(* CODESYS project Lark_Lubrication_AnandFeed.project
   Title: Lark_Lubrication_AnandFeed
   Version: 0.0.0.0

Project tree, tasks and I/O mapping:
  MyController : TM218LDA24DRN, Schneider Electric, order no. TM218LDA24DRN, version 4.0.1.26
    application Application
      libraries: Standard, * (System)
      task MAST (cyclic, interval 20 ms, priority 15, watchdog 100 ms x 1) calls POU
      function HiddenPOU [ST]
      global variables GVL
      program POU [FBD]
    Embedded Functions
      IO : IO, Schneider Electric, version 4.0.1.26
          input  iwIO_IW0 : WORD  // IW0
          input  Motor_Trip : BOOL  // IW0.I0
          input  Motor_ON_FB : BOOL  // IW0.I1
          input  Manual_Start : BOOL  // IW0.I2
          input  Manual_Stop : BOOL  // IW0.I3
          input  Manual_SS : BOOL  // IW0.I4
          input  Line2_SS : BOOL  // IW0.I5
          input  Tank_Empty_LS : BOOL  // IW0.I6
          input  Sensor1 : BOOL  // IW0.I7
          input  Sensor2 : BOOL  // IW0.I8
          output Motor_ON_CMD : BOOL  // QW0.Q0
          output Valve_On : BOOL  // QW0.Q3
          unmapped channels: QW0
      HSC : HSC, Schneider Electric, version 4.0.1.26
    Serial Line 1
      SoMachine_Network_Manager : SoMachine-Network Manager, Schneider Electric, version 4.0.0.2
    Serial Line 2
      Modbus_Manager : Modbus Manager, Schneider Electric, version 4.0.0.2
*)

// MyController/Application/GVL
VAR_GLOBAL
	
	Line1_On_Actual_Time AT %MD4 : DINT;
	Line1_Interval_Actual_Time AT %MD5 : DINT;
	
	Line2_On_Actual_Time AT %MD6 : DINT;
	Line2_Interval_Actual_Time AT %MD7 : DINT;
	
	Motor_Trip_IND AT %MX100.7: BOOL;
	Motor_On_IND AT %MX100.2: BOOL;
	Line1_On_CMD AT %MX100.4: BOOL;
	Line2_On_CMD AT %MX100.5: BOOL;
	Auto_SS AT %MX100.3: BOOL;
	TankEmptyLS_HMI AT %MX100.6: BOOL;
END_VAR

VAR_GLOBAL RETAIN
	Line1_SetTime AT %MD0 : DINT;
	Line1_IntervalTime AT %MD1 : DINT;
	
	Line2_SetTime AT %MD2 : DINT;
	Line2_IntervalTime AT %MD3 : DINT;
	
	Line1_Selected AT %MX100.0 : BOOL;
	Line2_Selected AT %MX100.1 : BOOL;
END_VAR

// MyController/Application/POU
PROGRAM POU
VAR
	TON_0: TON;
	SR_0: SR;
	R_TRIG_0: R_TRIG;
	SR_1: SR;
	Line1ON: BOOL;
	TON_1: TON;
	line1_SetTime_TIME: TIME;
	line1_On_ET_TIME: TIME;
	line1On_Elapsed: BOOL;
	line1_IntervalTime_TIME: TIME;
	line1_Int_ET_TIME: TIME;
	line1_Repeat: BOOL;
	RS_0: RS;
	Line2ON: BOOL;
	R_TRIG_1: R_TRIG;
	RS_1: RS;
	line2_Repeat: BOOL;
	TON_2: TON;
	line2_SetTime_TIME: TIME;
	line2_On_ET_TIME: TIME;
	line2On_Elapsed: BOOL;
	SR_2: SR;
	TON_3: TON;
	line2_IntervalTime_TIME: TIME;
	line2_Int_ET_TIME: TIME;
	RS_2: RS;
	Start_CMD: BOOL;
	Motor_ON_CMD_1: BOOL;
	Motor_ON_CMD_2: BOOL;
	TON_4: TON;
	test: BOOL;
END_VAR
VAR // added by the converter: edge detectors and wires of the graphical bodies
    _w1, _w2, _w3 : BOOL;
END_VAR

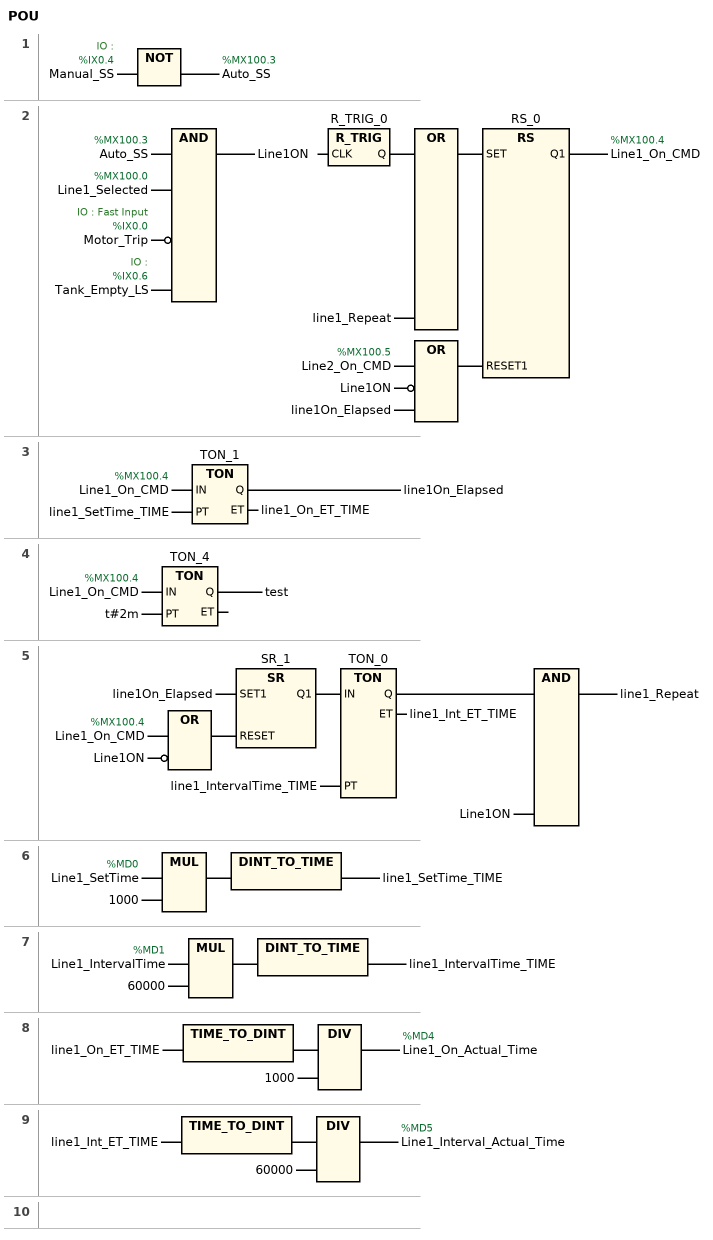
// NETWORK 1
//   Manual_SS: IO : | AT %IX0.4
//   Auto_SS: AT %MX100.3
Auto_SS := NOT Manual_SS;

// NETWORK 2
//   Auto_SS: AT %MX100.3
//   Line1_Selected: AT %MX100.0
//   Motor_Trip: IO : Fast Input | AT %IX0.0
//   Tank_Empty_LS: IO : | AT %IX0.6
//   Line2_On_CMD: AT %MX100.5
//   Line1_On_CMD: AT %MX100.4
_w1 := Auto_SS AND Line1_Selected AND NOT Motor_Trip AND Tank_Empty_LS;
Line1ON := _w1;
R_TRIG_0(CLK := _w1); // R_TRIG
RS_0(SET := R_TRIG_0.Q OR line1_Repeat, RESET1 := Line2_On_CMD OR NOT Line1ON OR line1On_Elapsed); // RS
Line1_On_CMD := RS_0.Q1;

// NETWORK 3
//   Line1_On_CMD: AT %MX100.4
TON_1(IN := Line1_On_CMD, PT := line1_SetTime_TIME, ET => line1_On_ET_TIME); // TON
line1On_Elapsed := TON_1.Q;

// NETWORK 4
//   Line1_On_CMD: AT %MX100.4
TON_4(IN := Line1_On_CMD, PT := t#2m); // TON
test := TON_4.Q;

// NETWORK 5
//   Line1_On_CMD: AT %MX100.4
SR_1(SET1 := line1On_Elapsed, RESET := Line1_On_CMD OR NOT Line1ON); // SR
TON_0(IN := SR_1.Q1, PT := line1_IntervalTime_TIME, ET => line1_Int_ET_TIME); // TON
line1_Repeat := TON_0.Q AND Line1ON;

// NETWORK 6
//   Line1_SetTime: AT %MD0
line1_SetTime_TIME := DINT_TO_TIME(Line1_SetTime * 1000);

// NETWORK 7
//   Line1_IntervalTime: AT %MD1
line1_IntervalTime_TIME := DINT_TO_TIME(Line1_IntervalTime * 60000);

// NETWORK 8
//   Line1_On_Actual_Time: AT %MD4
Line1_On_Actual_Time := TIME_TO_DINT(line1_On_ET_TIME) / 1000;

// NETWORK 9
//   Line1_Interval_Actual_Time: AT %MD5
Line1_Interval_Actual_Time := TIME_TO_DINT(line1_Int_ET_TIME) / 60000;

// NETWORK 10

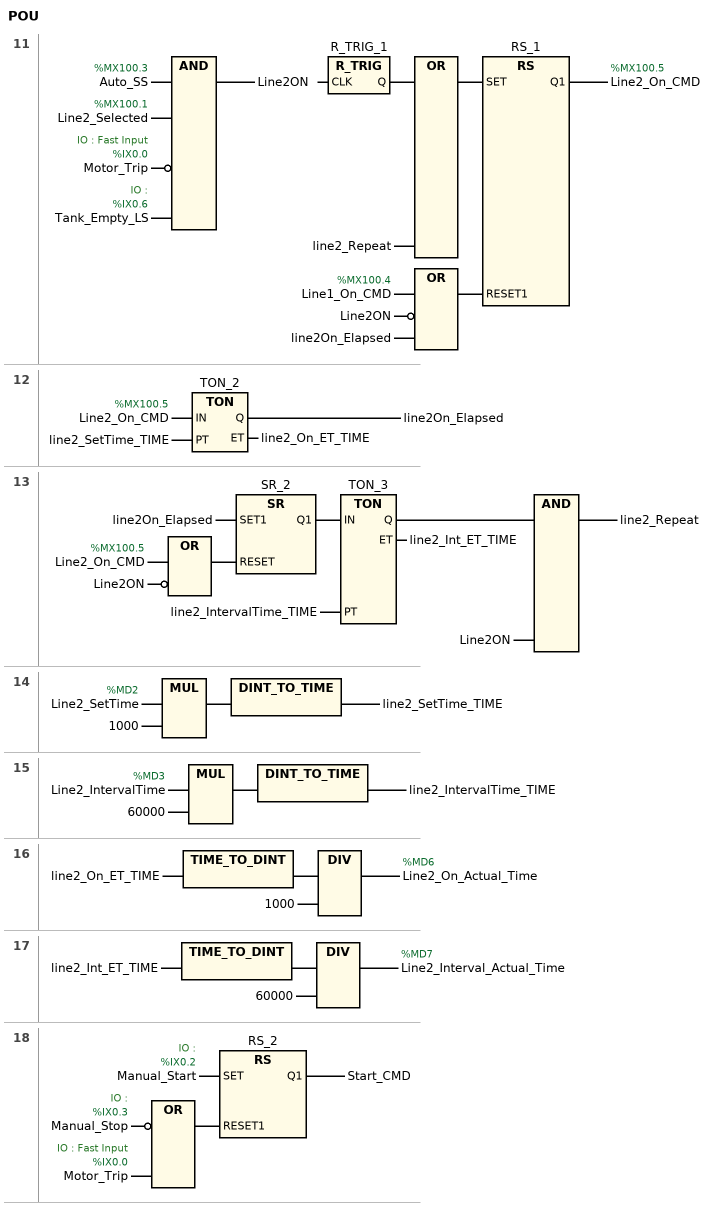
// NETWORK 11
//   Auto_SS: AT %MX100.3
//   Line2_Selected: AT %MX100.1
//   Motor_Trip: IO : Fast Input | AT %IX0.0
//   Tank_Empty_LS: IO : | AT %IX0.6
//   Line1_On_CMD: AT %MX100.4
//   Line2_On_CMD: AT %MX100.5
_w2 := Auto_SS AND Line2_Selected AND NOT Motor_Trip AND Tank_Empty_LS;
Line2ON := _w2;
R_TRIG_1(CLK := _w2); // R_TRIG
RS_1(SET := R_TRIG_1.Q OR line2_Repeat, RESET1 := Line1_On_CMD OR NOT Line2ON OR line2On_Elapsed); // RS
Line2_On_CMD := RS_1.Q1;

// NETWORK 12
//   Line2_On_CMD: AT %MX100.5
TON_2(IN := Line2_On_CMD, PT := line2_SetTime_TIME, ET => line2_On_ET_TIME); // TON
line2On_Elapsed := TON_2.Q;

// NETWORK 13
//   Line2_On_CMD: AT %MX100.5
SR_2(SET1 := line2On_Elapsed, RESET := Line2_On_CMD OR NOT Line2ON); // SR
TON_3(IN := SR_2.Q1, PT := line2_IntervalTime_TIME, ET => line2_Int_ET_TIME); // TON
line2_Repeat := TON_3.Q AND Line2ON;

// NETWORK 14
//   Line2_SetTime: AT %MD2
line2_SetTime_TIME := DINT_TO_TIME(Line2_SetTime * 1000);

// NETWORK 15
//   Line2_IntervalTime: AT %MD3
line2_IntervalTime_TIME := DINT_TO_TIME(Line2_IntervalTime * 60000);

// NETWORK 16
//   Line2_On_Actual_Time: AT %MD6
Line2_On_Actual_Time := TIME_TO_DINT(line2_On_ET_TIME) / 1000;

// NETWORK 17
//   Line2_Interval_Actual_Time: AT %MD7
Line2_Interval_Actual_Time := TIME_TO_DINT(line2_Int_ET_TIME) / 60000;

// NETWORK 18
//   Manual_Start: IO : | AT %IX0.2
//   Manual_Stop: IO : | AT %IX0.3
//   Motor_Trip: IO : Fast Input | AT %IX0.0
RS_2(SET := Manual_Start, RESET1 := NOT Manual_Stop OR Motor_Trip); // RS
Start_CMD := RS_2.Q1;

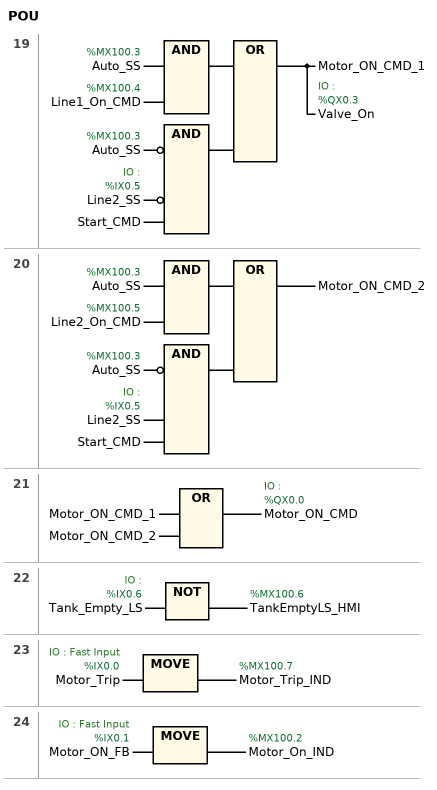
// NETWORK 19
//   Auto_SS: AT %MX100.3
//   Line1_On_CMD: AT %MX100.4
//   Line2_SS: IO : | AT %IX0.5
//   Valve_On: IO : | AT %QX0.3
_w3 := Auto_SS AND Line1_On_CMD OR NOT Auto_SS AND NOT Line2_SS AND Start_CMD;
Motor_ON_CMD_1 := _w3;
Valve_On := _w3;

// NETWORK 20
//   Auto_SS: AT %MX100.3
//   Line2_On_CMD: AT %MX100.5
//   Line2_SS: IO : | AT %IX0.5
Motor_ON_CMD_2 := Auto_SS AND Line2_On_CMD OR NOT Auto_SS AND Line2_SS AND Start_CMD;

// NETWORK 21
//   Motor_ON_CMD: IO : | AT %QX0.0
Motor_ON_CMD := Motor_ON_CMD_1 OR Motor_ON_CMD_2;

// NETWORK 22
//   Tank_Empty_LS: IO : | AT %IX0.6
//   TankEmptyLS_HMI: AT %MX100.6
TankEmptyLS_HMI := NOT Tank_Empty_LS;

// NETWORK 23
//   Motor_Trip: IO : Fast Input | AT %IX0.0
//   Motor_Trip_IND: AT %MX100.7
Motor_Trip_IND := Motor_Trip;

// NETWORK 24
//   Motor_ON_FB: IO : Fast Input | AT %IX0.1
//   Motor_On_IND: AT %MX100.2
Motor_On_IND := Motor_ON_FB;

END_PROGRAM

// MyController/Application/HiddenPOU
FUNCTION HiddenPOU : BOOL

VAR_INPUT
	pHiddenFunc: POINTER TO WORD;
END_VAR
VAR
	pRead: POINTER TO BYTE;
	pWrite: POINTER TO BYTE;
END_VAR

pRead := pHiddenFunc + 400;
pWrite := pHiddenFunc + 4400;
HiddenPOU := TRUE;

END_FUNCTION
